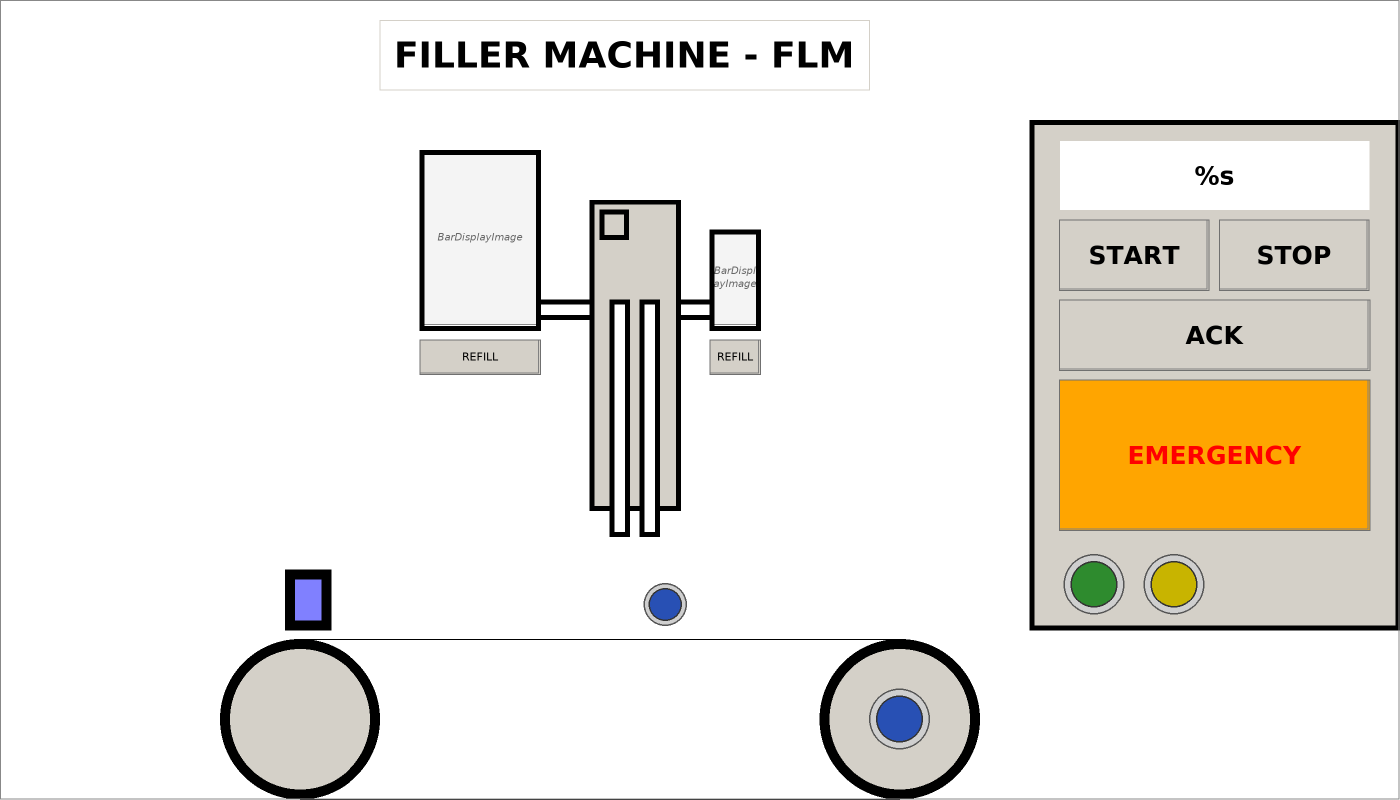
VISUALIZATION Visu  // 1401x801
    Rectangle (650,300 101x20), colour toggle: GVL_PLC.stFlmRawOut.bMint
    Rectangle (520,300 110x20), colour toggle: GVL_PLC.stFlmRawOut.bWater
    Rectangle (590,200 91x311), colour toggle: GVL_PLC.stFlmRawOut.bCorkingRotation
        p2738717112: (TO_REAL(GVL_PLC.stFlmRawOut.bCorkingVertical) * 50.0)
    Ellipse (220,640 160x160)
    Line (300,640) (900,640)
    Ellipse (820,640 160x160)
    Line (300,800) (900,800)
    Lamp1 (865,685 70x70), variable: GVL_PLC.stFlmRawOut.bConveyor, style: Lamp-Lamp1-Blue
    Rectangle (610,300 20x237), colour toggle: GVL_PLC.stFlmRawOut.bWater
    Rectangle (640,300 20x237), colour toggle: GVL_PLC.stFlmRawOut.bMint
    Lamp1 (640,580 51x50), variable: GVL_PLC.stFlmRawIn.bBottle, style: Lamp-Lamp1-Blue
    RoundedRectangle (285,570 46x61), invisible if: SIMU_MAIN.fPos > 100.0
        p3560616238: SIMU_MAIN.fPos * 5.0
    RoundedRectangle (1030,120 371x511)
    Button (1060,220 150x71), "START"
        tap GVL_PLC.stFlmRawIn.bStartButton
    Button (1220,220 150x71), "STOP"
        tap GVL_PLC.stFlmRawIn.bStopButton p1329445385=TRUE
    Textfield (1060,140 311x71), "%s", text variable: GVL_PLC.stFlmStatus.eStep
    Button (1060,300 311x71), "ACK"
        tap GVL_PLC.stFlmRawIn.bAckButton
    Button (1060,380 311x151), "EMERGENCY"
        toggle SIMU_MAIN.bEmergencyButton
    Group (710,230 51x101)
        BarDisplayImage (0,0 51x95), value: GVL_PLC.stFlmRawIn.nMintLevel, style: BarDisplayImage-Gray, scale format: %.1f, scale 0..32767
        Rectangle (0,0 51x101), colour toggle: GVL_PLC.stFlmRawOut.bCorkingRotation
    Group (420,150 121x181)
        BarDisplayImage (0,0 121x175), value: GVL_PLC.stFlmRawIn.nWaterLevel, style: BarDisplayImage-Gray, scale format: %.1f, scale 0..32767
        Rectangle (0,0 121x181), colour toggle: GVL_PLC.stFlmRawOut.bCorkingRotation
    RoundedRectangle (600,210 29x30), colour toggle: GVL_PLC.stFlmRawIn.bCorkingRotationLimitSwitch
        p2738717112: (TO_REAL(GVL_PLC.stFlmRawOut.bCorkingVertical) * 50.0)
    Button (420,340 121x35), "REFILL"
        tap SIMU_MAIN.bRefillWater
    Button (710,340 51x35), "REFILL"
        tap SIMU_MAIN.bRefillMint
    Lamp1 (1060,550 70x70), variable: GVL_PLC.stFlmRawOut.bGreen, style: Lamp-Lamp1-Green
    Lamp1 (1140,550 70x70), variable: GVL_PLC.stFlmRawOut.bYellow, style: Lamp-Lamp1-Yellow
    Textfield (380,20 490x70), "FILLER MACHINE - FLM"
END_VISUALIZATION

(* stored: Version 1.1.0.1, ProductVersion 3.1.4024.12
   Visu Visu: Id {79eb8f98-2db4-4b83-985c-94485c8e1a1b} *)
